# EPICS IOC start-up script: iocsh/dtl-tuners-noalias.iocsh
##############################################################################
############ Startup File for DTL Tuners System
############
############ Author: Maurizio Montis || INFN-LNL
############ Mail:   maurizio.montis@lnl.infn.it
############
##############################################################################

##############################################################################
############ Environment

###
############ Configuration
############ Set the values in order to proper configure the application
############
###
#
### Communication
# Ethercat Master Index
epicsEnvSet("MASTER_ID", "0")

### Application
# IOC application name
epicsEnvSet("IOC", "DTL-000")
# Modules version
epicsEnvSet("ECMCCFG_VERSION", "6.2.0")
epicsEnvSet("ECMC_VERSION", "6.2.1")
epicsEnvSet("STREAM_VERSION", "2.8.10")
# Axis configuration
epicsEnvSet("DTL_AXIS_PATH", "/home/iocuser/e3/e3-dtlTuners/cfg")

#
############ End of Configuration part
#

### Standard Configuration - DO NOT MODIFY
#
epicsEnvSet("ECMC_CONFIG_ROOT",     "${E3_SITEMODS_PATH}/ecmccfg/${ECMCCFG_VERSION}/")
epicsEnvSet("ECMC_CONFIG_DB",       "${ECMC_CONFIG_ROOT}db/")
epicsEnvSet("SCRIPTEXEC",           "${SCRIPTEXEC=iocshLoad}")
epicsEnvSet("STREAM_PROTOCOL_PATH", "${STREAM_PROTOCOL_PATH=""}:${ECMC_CONFIG_ROOT}:${ECMC_CONFIG_DB}")
epicsEnvSet("SM_PREFIX",            "${IOC}:")

##############################################################################
############ Modules Required

require ecmccfg, ${ECMCCFG_VERSION}
require ecmc, ${ECMC_VERSION}
require stream, ${STREAM_VERSION}

##############################################################################
############ Application Initialization

${SCRIPTEXEC} "${ECMC_CONFIG_ROOT}${INIT=initAll}.cmd"

##############################################################################
############ EtherCAT Master Configuration

${SCRIPTEXEC} "${ECMC_CONFIG_ROOT}addMaster.cmd", "MASTER_ID=${MASTER_ID}"

##############################################################################
############ EtherCAT Slaves Configuration

# - Module EK1100
${SCRIPTEXEC} "${ECMC_CONFIG_ROOT}addSlave.cmd", "HW_DESC=EK1100, SLAVE_ID=0"

# - Module EL7047
${SCRIPTEXEC} "${ECMC_CONFIG_ROOT}addSlave.cmd", "HW_DESC=EL7047, SLAVE_ID=4"
${SCRIPTEXEC} "${ECMC_CONFIG_ROOT}applySlaveConfig.cmd",   "CONFIG=-Motor-Leadshine-57HS09"

# - Module EL3255
${SCRIPTEXEC} "${ECMC_CONFIG_ROOT}addSlave.cmd", "HW_DESC=EL3255, SLAVE_ID=3"

# - Module EL2124
#${SCRIPTEXEC} "${ECMC_CONFIG_ROOT}addSlave.cmd", "HW_DESC=EL2124, SLAVE_ID=3"

##############################################################################
############# Apply Configuration

${SCRIPTEXEC} "${ECMC_CONFIG_ROOT}applyConfig.cmd"

##############################################################################
############ Axis Configuration

# - Axis T1M1
epicsEnvSet("DEV",      "AXIS")
${SCRIPTEXEC} "${ECMC_CONFIG_ROOT}configureAxis.cmd", "CONFIG=${DTL_AXIS_PATH}/axis_T0M0"

# Apply Axes Configuration - REQUIRED
${SCRIPTEXEC} "${ECMC_CONFIG_ROOT}applyConfig.cmd"

##############################################################################
############ Go Active

${SCRIPTEXEC} "${ECMC_CONFIG_ROOT}setAppMode.cmd"
